// TIA Portal V19 export
VAR_GLOBAL   // PLC tag table "LB311"
   LB311_DeadMan_Ch2 AT %I1300.7 : Bool;   // 250DI7 - 264SB1
   LB311_DeadMan_Ch1 AT %I1300.3 : Bool;   // 250DI3 - 264SB1
   LB311_Bordatrice_Pb_Indietro AT %I273.3 : Bool;   // 352SB1
   LB311_Bordatrice_Pb_Avanti AT %I273.4 : Bool;   // 352SB2
END_VAR
